// Mitsubishi GX Works2 project: solEx1   PLC: Q03UDV

PROGRAM MAIN
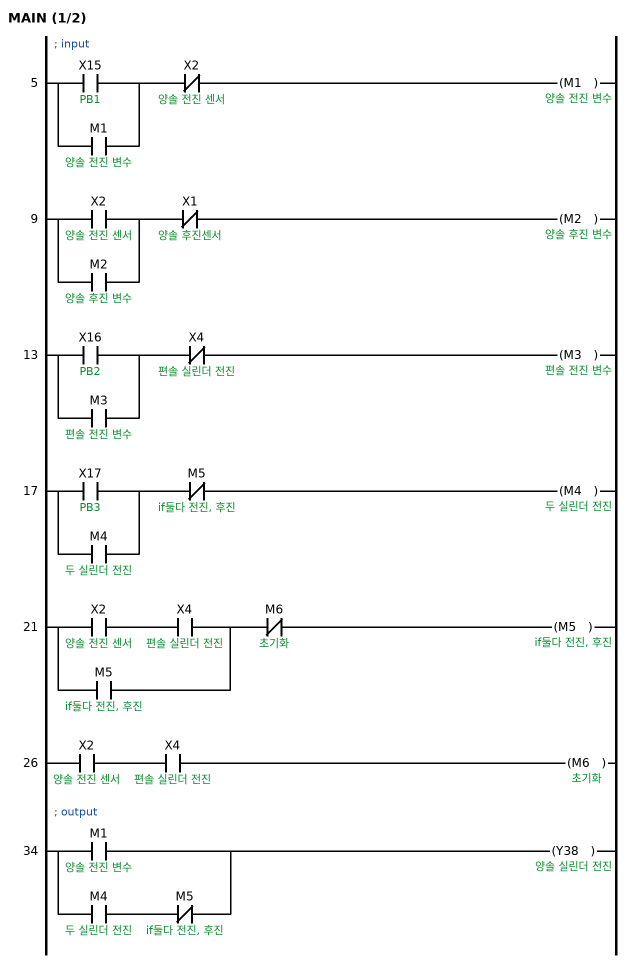
; input
5     LD      X15  ; PB1
      OR      M1  ; 양솔 전진 변수
      ANI     X2  ; 양솔 전진 센서
      OUT     M1  ; 양솔 전진 변수
9     LD      X2  ; 양솔 전진 센서
      OR      M2  ; 양솔 후진 변수
      ANI     X1  ; 양솔 후진센서
      OUT     M2  ; 양솔 후진 변수
13    LD      X16  ; PB2
      OR      M3  ; 편솔 전진 변수
      ANI     X4  ; 편솔 실린더 전진
      OUT     M3  ; 편솔 전진 변수
17    LD      X17  ; PB3
      OR      M4  ; 두 실린더 전진
      ANI     M5  ; if둘다 전진, 후진
      OUT     M4  ; 두 실린더 전진
21    LD      X2  ; 양솔 전진 센서
      AND     X4  ; 편솔 실린더 전진
      OR      M5  ; if둘다 전진, 후진
      ANI     M6  ; 초기화
      OUT     M5  ; if둘다 전진, 후진
26    LD      X2  ; 양솔 전진 센서
      AND     X4  ; 편솔 실린더 전진
      OUT     M6  ; 초기화
; output
34    LD      M1  ; 양솔 전진 변수
      LD      M4  ; 두 실린더 전진
      ANI     M5  ; if둘다 전진, 후진
      ORB
      OUT     Y38  ; 양솔 실린더 전진
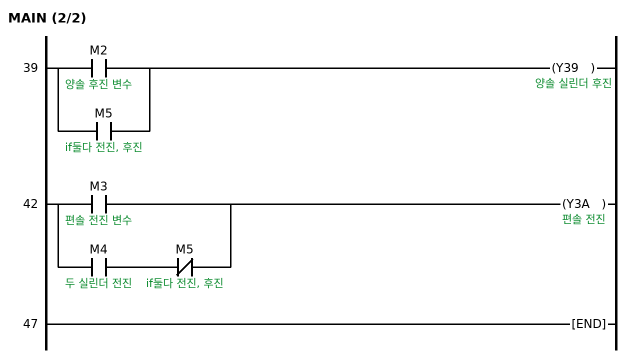
39    LD      M2  ; 양솔 후진 변수
      OR      M5  ; if둘다 전진, 후진
      OUT     Y39  ; 양솔 실린더 후진
42    LD      M3  ; 편솔 전진 변수
      LD      M4  ; 두 실린더 전진
      ANI     M5  ; if둘다 전진, 후진
      ORB
      OUT     Y3A  ; 편솔 전진
47    END
END_PROGRAM

// device comments not shown above
X3  ; 편솔 후진
